TYPE MachineSts_typ :
STRUCT
	Enabled	: BOOL;
	Running	: BOOL;
	Error	: BOOL;
	State	: MachineState_enum;
END_STRUCT
END_TYPE

(* stored: Version 1.1.0.1, ProductVersion 3.1.4026.8
   DUT MachineSts_typ: Id {d64e0d58-f4a7-0e1c-0076-17a9efd6aafb} *)
